// TIA Portal V17 export
// export: Created 2023-02-14T02:49:25.7164251Z, ExportSetting WithDefaults, DisplayName Totally Integrated Automation Portal, DisplayVersion V17, DisplayName TIA Portal Openness, DisplayVersion V17, DisplayName TIA Portal Teamcenter Gateway, DisplayVersion V17, DisplayName TIA Portal Version Control Interface, DisplayVersion V17, DisplayName SINAMICS Startdrive Advanced, DisplayVersion V17, DisplayName SINAMICS Startdrive G130, G150, S120, S150, SINAMICS MV, S210, DisplayVersion V17, DisplayName SINAMICS Startdrive G110M, G120, G120C, G120D, G120P, G115D, DisplayVersion V17, DisplayName STEP 7 Professional, DisplayVersion V17, DisplayName STEP 7 Safety, DisplayVersion V17, DisplayName WinCC Professional, DisplayVersion V17
FUNCTION_BLOCK "IO_Valve_Blend21"   // FB25, LAD
{ S7_Optimized_Access := 'FALSE' }
VERSION : 0.1
// stored: AutoNumber true, IsIECCheckEnabled false, SetENOAutomatically false, UDAEnableTagReadback false
   VAR_INPUT
      "lock 1" : Bool;
      "lock 2" : Bool;
      "lock 3" : Bool;
      "lock 4" : Bool;
      init : Bool;
      reset : Bool;
      testing : Bool;
   END_VAR
   VAR
      "AV-21.01" : "Valve";
      "AV-21.02" : "Valve";
      "AV-21.03" : "Valve";
      "AV-21.04" : "Valve";
      "AV-21.05" : "Valve";
      "AV-21.06" : "Valve";
      "AV-21.07" : "Valve";
      "AV-21.08" : "Valve";
      "AV-21.09" : "Valve";
      "AV-21.10" : "Valve";
      "AV-21.11" : "Valve";
      "AV-21.21" : "Valve";
      "AV-21.22" : "Valve";
      "AV-21.23" : "Valve";
      "AV-21.24" : "Valve";
      "AV-21.25" : "Valve";
      "AV-21.26" : "Valve";
      "AV-21.27" : "Valve";
      "AV-21.28" : "Valve";
      "AV-21.29" : "Valve";
      "AV-21.30" : "Valve";
      "AV-21.31" : "Valve";
      "AV-21.32" : "Valve";
      "AV-21.33" : "Valve";
      "AV-21.34" : "Valve";
      "AV-21.35" : "Valve";
      "AV-21.41" : "Valve";
      "AV-21.42" : "Valve";
   END_VAR
BEGIN

REGION Network 1 (SCL): FB OPEN AND CLOSE VALVE T-21
   IF #testing THEN
       // Statement section IF
       #"AV-21.01".FB_OPEN := #"AV-21.01".QCMD_OP;
       #"AV-21.01".FB_CLOSE := NOT #"AV-21.01".QCMD_OP;
       #"AV-21.02".FB_OPEN := #"AV-21.02".QCMD_OP;
       #"AV-21.02".FB_CLOSE := NOT #"AV-21.02".QCMD_OP;
       #"AV-21.03".FB_OPEN := #"AV-21.03".QCMD_OP;
       #"AV-21.03".FB_CLOSE := NOT #"AV-21.03".QCMD_OP;
       #"AV-21.04".FB_OPEN := #"AV-21.04".QCMD_OP;
       #"AV-21.04".FB_CLOSE := NOT #"AV-21.04".QCMD_OP;
       #"AV-21.05".FB_OPEN := #"AV-21.05".QCMD_OP;
       #"AV-21.05".FB_CLOSE := NOT #"AV-21.05".QCMD_OP;
       #"AV-21.06".FB_OPEN := #"AV-21.06".QCMD_OP;
       #"AV-21.06".FB_CLOSE := NOT #"AV-21.06".QCMD_OP;
       #"AV-21.07".FB_OPEN := #"AV-21.07".QCMD_OP;
       #"AV-21.07".FB_CLOSE := NOT #"AV-21.07".QCMD_OP;
       #"AV-21.08".FB_OPEN := #"AV-21.08".QCMD_OP;
       #"AV-21.08".FB_CLOSE := NOT #"AV-21.08".QCMD_OP;
       #"AV-21.09".FB_OPEN := #"AV-21.09".QCMD_OP;
       #"AV-21.09".FB_CLOSE := NOT #"AV-21.09".QCMD_OP;
       #"AV-21.10".FB_OPEN := #"AV-21.10".QCMD_OP;
       #"AV-21.10".FB_CLOSE := NOT #"AV-21.10".QCMD_OP;
       #"AV-21.11".FB_OPEN := #"AV-21.11".QCMD_OP;
       #"AV-21.11".FB_CLOSE := NOT #"AV-21.11".QCMD_OP;
       #"AV-21.21".FB_OPEN := #"AV-21.21".QCMD_OP;
       #"AV-21.21".FB_CLOSE := NOT #"AV-21.21".QCMD_OP;
       #"AV-21.22".FB_OPEN := #"AV-21.22".QCMD_OP;
       #"AV-21.22".FB_CLOSE := NOT #"AV-21.22".QCMD_OP;
       #"AV-21.23".FB_OPEN := #"AV-21.23".QCMD_OP;
       #"AV-21.23".FB_CLOSE := NOT #"AV-21.23".QCMD_OP;
       #"AV-21.24".FB_OPEN := #"AV-21.24".QCMD_OP;
       #"AV-21.24".FB_CLOSE := NOT #"AV-21.24".QCMD_OP;
       #"AV-21.25".FB_OPEN := #"AV-21.25".QCMD_OP;
       #"AV-21.25".FB_CLOSE := NOT #"AV-21.25".QCMD_OP;
       #"AV-21.26".FB_OPEN := #"AV-21.26".QCMD_OP;
       #"AV-21.26".FB_CLOSE := NOT #"AV-21.26".QCMD_OP;
       #"AV-21.27".FB_OPEN := #"AV-21.27".QCMD_OP;
       #"AV-21.27".FB_CLOSE := NOT #"AV-21.27".QCMD_OP;
       #"AV-21.28".FB_OPEN := #"AV-21.28".QCMD_OP;
       #"AV-21.28".FB_CLOSE := NOT #"AV-21.28".QCMD_OP;
       #"AV-21.29".FB_OPEN := #"AV-21.29".QCMD_OP;
       #"AV-21.29".FB_CLOSE := NOT #"AV-21.29".QCMD_OP;
       #"AV-21.30".FB_OPEN := #"AV-21.30".QCMD_OP;
       #"AV-21.30".FB_CLOSE := NOT #"AV-21.30".QCMD_OP;
       #"AV-21.31".FB_OPEN := #"AV-21.31".QCMD_OP;
       #"AV-21.31".FB_CLOSE := NOT #"AV-21.31".QCMD_OP;
       #"AV-21.32".FB_OPEN := #"AV-21.32".QCMD_OP;
       #"AV-21.32".FB_CLOSE := NOT #"AV-21.32".QCMD_OP;
       #"AV-21.33".FB_OPEN := #"AV-21.33".QCMD_OP;
       #"AV-21.33".FB_CLOSE := NOT #"AV-21.33".QCMD_OP;
       #"AV-21.34".FB_OPEN := #"AV-21.34".QCMD_OP;
       #"AV-21.34".FB_CLOSE := NOT #"AV-21.34".QCMD_OP;
       #"AV-21.35".FB_OPEN := #"AV-21.35".QCMD_OP;
       #"AV-21.35".FB_CLOSE := NOT #"AV-21.35".QCMD_OP;
       #"AV-21.41".FB_OPEN := #"AV-21.41".QCMD_OP;
       #"AV-21.41".FB_CLOSE := NOT #"AV-21.41".QCMD_OP;
       #"AV-21.42".FB_OPEN := #"AV-21.42".QCMD_OP;
       #"AV-21.42".FB_CLOSE := NOT #"AV-21.42".QCMD_OP;
   ELSE
       // Statement section ELSE
       #"AV-21.01".FB_OPEN := #"AV-21.01".QCMD_OP;
       #"AV-21.01".FB_CLOSE := NOT #"AV-21.01".QCMD_OP;
       #"AV-21.02".FB_OPEN := NOT "ZSC-21.02";
       #"AV-21.02".FB_CLOSE := "ZSC-21.02";
       #"AV-21.03".FB_OPEN := NOT "ZSC-21.03";
       #"AV-21.03".FB_CLOSE := "ZSC-21.03";
       #"AV-21.04".FB_OPEN := #"AV-21.04".QCMD_OP;
       #"AV-21.04".FB_CLOSE := NOT #"AV-21.04".QCMD_OP;
       #"AV-21.05".FB_OPEN := NOT "ZSC-21.05";
       #"AV-21.05".FB_CLOSE := "ZSC-21.05";
       #"AV-21.06".FB_OPEN := NOT "ZSC-21.06";
       #"AV-21.06".FB_CLOSE := "ZSC-21.06";
       #"AV-21.07".FB_OPEN := #"AV-21.07".QCMD_OP;
       #"AV-21.07".FB_CLOSE := NOT #"AV-21.07".QCMD_OP;
       #"AV-21.08".FB_OPEN := NOT "ZSC-21.08";
       #"AV-21.08".FB_CLOSE := "ZSC-21.08";
       #"AV-21.09".FB_OPEN := NOT "ZSC-21.09";
       #"AV-21.09".FB_CLOSE := "ZSC-21.09";
       #"AV-21.10".FB_OPEN := #"AV-21.10".QCMD_OP;
       #"AV-21.10".FB_CLOSE := NOT #"AV-21.10".QCMD_OP;
       #"AV-21.11".FB_OPEN := NOT "ZSC-21.11";
       #"AV-21.11".FB_CLOSE := "ZSC-21.11";
       #"AV-21.21".FB_OPEN := NOT "ZSC-21.21";
       #"AV-21.21".FB_CLOSE := "ZSC-21.21";
       #"AV-21.22".FB_OPEN := #"AV-21.22".QCMD_OP;
       #"AV-21.22".FB_CLOSE := NOT #"AV-21.22".QCMD_OP;
       #"AV-21.23".FB_OPEN := NOT "ZSC-21.23";
       #"AV-21.23".FB_CLOSE := "ZSC-21.23";
       #"AV-21.24".FB_OPEN := NOT "ZSC-21.24";
       #"AV-21.24".FB_CLOSE := "ZSC-21.24";
       #"AV-21.25".FB_OPEN := NOT "ZSC-21.25";
       #"AV-21.25".FB_CLOSE := "ZSC-21.25";
       #"AV-21.26".FB_OPEN := #"AV-21.26".QCMD_OP;
       #"AV-21.26".FB_CLOSE := NOT #"AV-21.26".QCMD_OP;
       #"AV-21.27".FB_OPEN := NOT "ZSC-21.27";
       #"AV-21.27".FB_CLOSE := "ZSC-21.27";
       #"AV-21.28".FB_OPEN := NOT "ZSC-21.28";
       #"AV-21.28".FB_CLOSE := "ZSC-21.28";
       #"AV-21.29".FB_OPEN := #"AV-21.29".QCMD_OP;
       #"AV-21.29".FB_CLOSE := NOT #"AV-21.29".QCMD_OP;
       #"AV-21.30".FB_OPEN := #"AV-21.30".QCMD_OP;
       #"AV-21.30".FB_CLOSE := NOT #"AV-21.30".QCMD_OP;
       #"AV-21.31".FB_OPEN := NOT "ZSC-21.31";
       #"AV-21.31".FB_CLOSE := "ZSC-21.31";
       #"AV-21.32".FB_OPEN := NOT "ZSC-21.32";
       #"AV-21.32".FB_CLOSE := "ZSC-21.32";
       #"AV-21.33".FB_OPEN := NOT "ZSC-21.33";
       #"AV-21.33".FB_CLOSE := "ZSC-21.33";
       #"AV-21.34".FB_OPEN := NOT "ZSC-21.34";
       #"AV-21.34".FB_CLOSE := "ZSC-21.34";
       #"AV-21.35".FB_OPEN := NOT "ZSC-21.35";
       #"AV-21.35".FB_CLOSE := "ZSC-21.35";
       #"AV-21.41".FB_OPEN := #"AV-21.41".QCMD_OP;
       #"AV-21.41".FB_CLOSE := NOT #"AV-21.41".QCMD_OP;
       #"AV-21.42".FB_OPEN := #"AV-21.42".QCMD_OP;
       #"AV-21.42".FB_CLOSE := NOT #"AV-21.42".QCMD_OP;
   END_IF;
END_REGION

NETWORK
TITLE = FB MONITORING TIME VALVE T-21
// FB OPEN TIME
      L     T#20s;
      T     #"AV-21.01".MON_T;
      T     #"AV-21.02".MON_T;
      T     #"AV-21.03".MON_T;
      T     #"AV-21.04".MON_T;
      T     #"AV-21.05".MON_T;
      T     #"AV-21.06".MON_T;
      T     #"AV-21.07".MON_T;
      T     #"AV-21.08".MON_T;
      T     #"AV-21.09".MON_T;
      T     #"AV-21.10".MON_T;
      T     #"AV-21.11".MON_T;
      T     #"AV-21.21".MON_T;
      T     #"AV-21.22".MON_T;
      T     #"AV-21.23".MON_T;
      T     #"AV-21.24".MON_T;
      T     #"AV-21.25".MON_T;
      T     #"AV-21.26".MON_T;
      T     #"AV-21.27".MON_T;
      T     #"AV-21.28".MON_T;
      T     #"AV-21.29".MON_T;
      T     #"AV-21.30".MON_T;
      T     #"AV-21.31".MON_T;
      T     #"AV-21.32".MON_T;
      T     #"AV-21.33".MON_T;
      T     #"AV-21.34".MON_T;
      T     #"AV-21.35".MON_T;
      T     #"AV-21.41".MON_T;
      T     #"AV-21.42".MON_T;

// FB CLOSE TIME
      L     T#20s;
      T     #"AV-21.01".MON_T_CLOSE;
      T     #"AV-21.02".MON_T_CLOSE;
      T     #"AV-21.03".MON_T_CLOSE;
      T     #"AV-21.04".MON_T_CLOSE;
      T     #"AV-21.05".MON_T_CLOSE;
      T     #"AV-21.06".MON_T_CLOSE;
      T     #"AV-21.07".MON_T_CLOSE;
      T     #"AV-21.08".MON_T_CLOSE;
      T     #"AV-21.09".MON_T_CLOSE;
      T     #"AV-21.10".MON_T_CLOSE;
      T     #"AV-21.11".MON_T_CLOSE;
      T     #"AV-21.21".MON_T_CLOSE;
      T     #"AV-21.22".MON_T_CLOSE;
      T     #"AV-21.23".MON_T_CLOSE;
      T     #"AV-21.24".MON_T_CLOSE;
      T     #"AV-21.25".MON_T_CLOSE;
      T     #"AV-21.26".MON_T_CLOSE;
      T     #"AV-21.27".MON_T_CLOSE;
      T     #"AV-21.28".MON_T_CLOSE;
      T     #"AV-21.29".MON_T_CLOSE;
      T     #"AV-21.30".MON_T_CLOSE;
      T     #"AV-21.31".MON_T_CLOSE;
      T     #"AV-21.32".MON_T_CLOSE;
      T     #"AV-21.33".MON_T_CLOSE;
      T     #"AV-21.34".MON_T_CLOSE;
      T     #"AV-21.35".MON_T_CLOSE;
      T     #"AV-21.41".MON_T_CLOSE;
      T     #"AV-21.42".MON_T_CLOSE;


REGION Network 3: AV-21.01
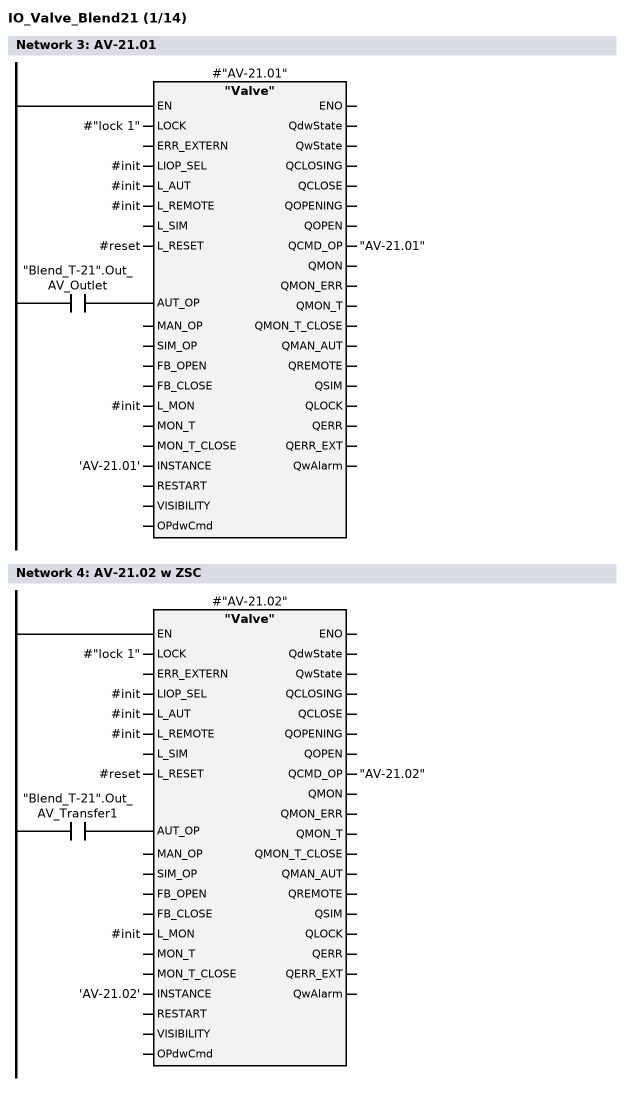
   RUNG wire#powerrail
      #"AV-21.01"(AUT_OP := wire#w1, LOCK := #"lock 1", ERR_EXTERN :=, LIOP_SEL := #init, L_AUT := #init, L_REMOTE := #init, L_SIM :=, L_RESET := #reset, MAN_OP :=, SIM_OP :=, FB_OPEN :=, FB_CLOSE :=, L_MON := #init, MON_T :=, MON_T_CLOSE :=, INSTANCE := 'AV-21.01', RESTART :=, VISIBILITY :=, OPdwCmd :=, QdwState =>, QwState =>, QCLOSING =>, QCLOSE =>, QOPENING =>, QOPEN =>, QCMD_OP => "AV-21.01", QMON =>, QMON_ERR =>, QMON_T =>, QMON_T_CLOSE =>, QMAN_AUT =>, QREMOTE =>, QSIM =>, QLOCK =>, QERR =>, QERR_EXT =>, QwAlarm =>)
   END_RUNG
   RUNG wire#powerrail
      Contact( "Blend_T-21".Out_AV_Outlet )
   END_RUNG wire#w1
   // the same network as SCL:
   #"AV-21.01"(LOCK := #"lock 1",   // "Valve"
               LIOP_SEL := #init,
               L_AUT := #init,
               L_REMOTE := #init,
               L_RESET := #reset,
               AUT_OP := "Blend_T-21".Out_AV_Outlet,
               L_MON := #init,
               INSTANCE := 'AV-21.01',
               QCMD_OP => "AV-21.01");
END_REGION

REGION Network 4: AV-21.02 w ZSC
   RUNG wire#powerrail
      #"AV-21.02"(AUT_OP := wire#w1, LOCK := #"lock 1", ERR_EXTERN :=, LIOP_SEL := #init, L_AUT := #init, L_REMOTE := #init, L_SIM :=, L_RESET := #reset, MAN_OP :=, SIM_OP :=, FB_OPEN :=, FB_CLOSE :=, L_MON := #init, MON_T :=, MON_T_CLOSE :=, INSTANCE := 'AV-21.02', RESTART :=, VISIBILITY :=, OPdwCmd :=, QdwState =>, QwState =>, QCLOSING =>, QCLOSE =>, QOPENING =>, QOPEN =>, QCMD_OP => "AV-21.02", QMON =>, QMON_ERR =>, QMON_T =>, QMON_T_CLOSE =>, QMAN_AUT =>, QREMOTE =>, QSIM =>, QLOCK =>, QERR =>, QERR_EXT =>, QwAlarm =>)
   END_RUNG
   RUNG wire#powerrail
      Contact( "Blend_T-21".Out_AV_Transfer1 )
   END_RUNG wire#w1
   // the same network as SCL:
   #"AV-21.02"(LOCK := #"lock 1",   // "Valve"
               LIOP_SEL := #init,
               L_AUT := #init,
               L_REMOTE := #init,
               L_RESET := #reset,
               AUT_OP := "Blend_T-21".Out_AV_Transfer1,
               L_MON := #init,
               INSTANCE := 'AV-21.02',
               QCMD_OP => "AV-21.02");
END_REGION

REGION Network 5: AV-21.03 w ZSC
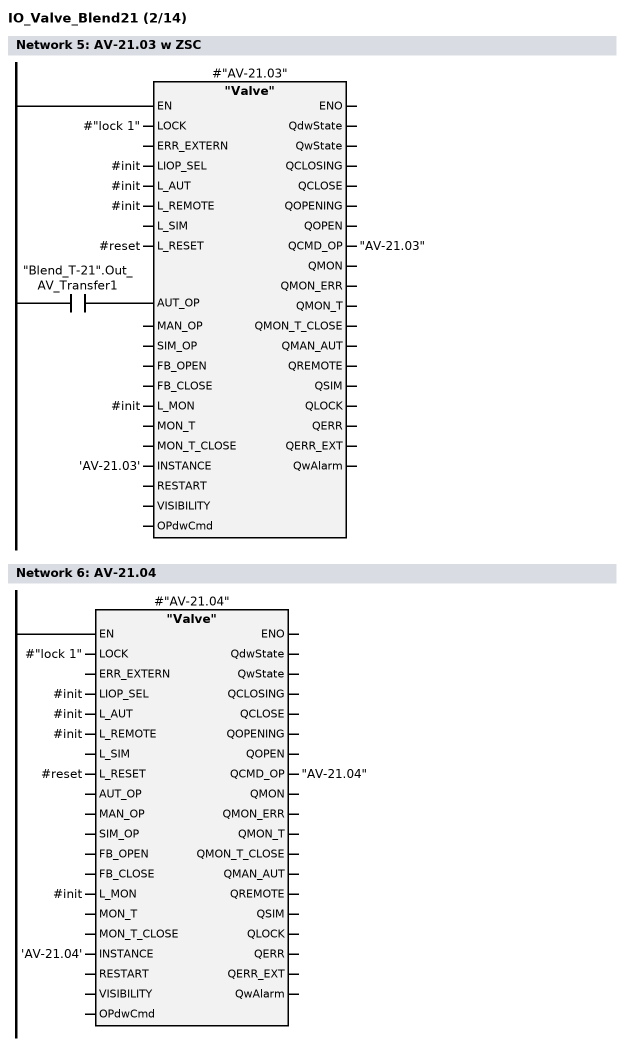
   RUNG wire#powerrail
      #"AV-21.03"(AUT_OP := wire#w1, LOCK := #"lock 1", ERR_EXTERN :=, LIOP_SEL := #init, L_AUT := #init, L_REMOTE := #init, L_SIM :=, L_RESET := #reset, MAN_OP :=, SIM_OP :=, FB_OPEN :=, FB_CLOSE :=, L_MON := #init, MON_T :=, MON_T_CLOSE :=, INSTANCE := 'AV-21.03', RESTART :=, VISIBILITY :=, OPdwCmd :=, QdwState =>, QwState =>, QCLOSING =>, QCLOSE =>, QOPENING =>, QOPEN =>, QCMD_OP => "AV-21.03", QMON =>, QMON_ERR =>, QMON_T =>, QMON_T_CLOSE =>, QMAN_AUT =>, QREMOTE =>, QSIM =>, QLOCK =>, QERR =>, QERR_EXT =>, QwAlarm =>)
   END_RUNG
   RUNG wire#powerrail
      Contact( "Blend_T-21".Out_AV_Transfer1 )
   END_RUNG wire#w1
   // the same network as SCL:
   #"AV-21.03"(LOCK := #"lock 1",   // "Valve"
               LIOP_SEL := #init,
               L_AUT := #init,
               L_REMOTE := #init,
               L_RESET := #reset,
               AUT_OP := "Blend_T-21".Out_AV_Transfer1,
               L_MON := #init,
               INSTANCE := 'AV-21.03',
               QCMD_OP => "AV-21.03");
END_REGION

REGION Network 6: AV-21.04
   RUNG wire#powerrail
      #"AV-21.04"(LOCK := #"lock 1", ERR_EXTERN :=, LIOP_SEL := #init, L_AUT := #init, L_REMOTE := #init, L_SIM :=, L_RESET := #reset, AUT_OP :=, MAN_OP :=, SIM_OP :=, FB_OPEN :=, FB_CLOSE :=, L_MON := #init, MON_T :=, MON_T_CLOSE :=, INSTANCE := 'AV-21.04', RESTART :=, VISIBILITY :=, OPdwCmd :=, QdwState =>, QwState =>, QCLOSING =>, QCLOSE =>, QOPENING =>, QOPEN =>, QCMD_OP => "AV-21.04", QMON =>, QMON_ERR =>, QMON_T =>, QMON_T_CLOSE =>, QMAN_AUT =>, QREMOTE =>, QSIM =>, QLOCK =>, QERR =>, QERR_EXT =>, QwAlarm =>)
   END_RUNG
   // the same network as SCL:
   #"AV-21.04"(LOCK := #"lock 1",   // "Valve"
               LIOP_SEL := #init,
               L_AUT := #init,
               L_REMOTE := #init,
               L_RESET := #reset,
               L_MON := #init,
               INSTANCE := 'AV-21.04',
               QCMD_OP => "AV-21.04");
END_REGION

REGION Network 7: AV-21.05 w ZSC
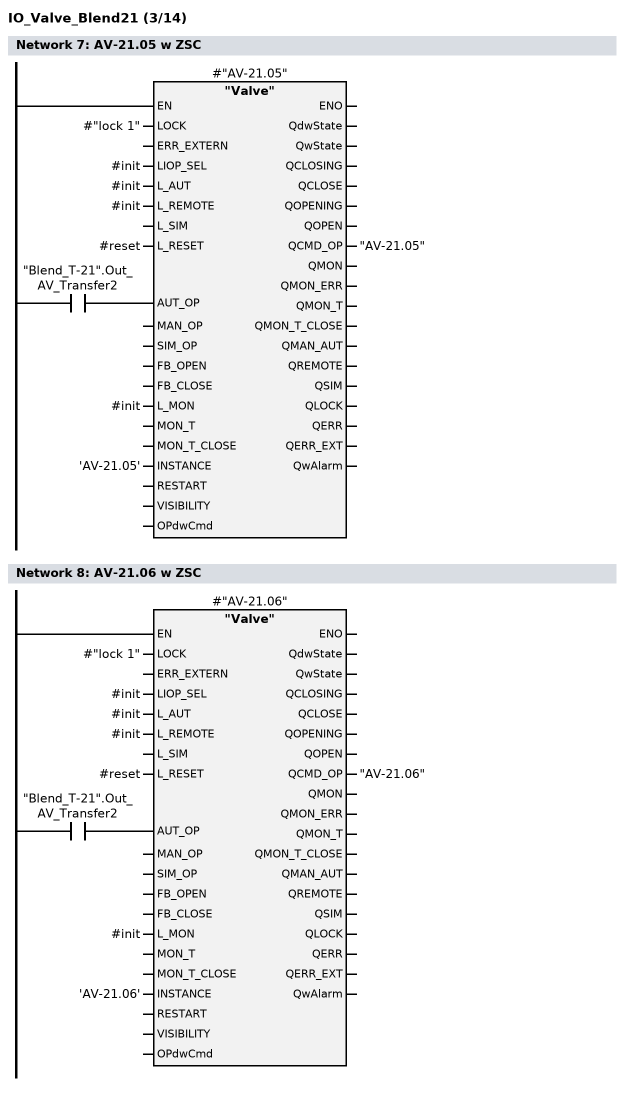
   RUNG wire#powerrail
      #"AV-21.05"(AUT_OP := wire#w1, LOCK := #"lock 1", ERR_EXTERN :=, LIOP_SEL := #init, L_AUT := #init, L_REMOTE := #init, L_SIM :=, L_RESET := #reset, MAN_OP :=, SIM_OP :=, FB_OPEN :=, FB_CLOSE :=, L_MON := #init, MON_T :=, MON_T_CLOSE :=, INSTANCE := 'AV-21.05', RESTART :=, VISIBILITY :=, OPdwCmd :=, QdwState =>, QwState =>, QCLOSING =>, QCLOSE =>, QOPENING =>, QOPEN =>, QCMD_OP => "AV-21.05", QMON =>, QMON_ERR =>, QMON_T =>, QMON_T_CLOSE =>, QMAN_AUT =>, QREMOTE =>, QSIM =>, QLOCK =>, QERR =>, QERR_EXT =>, QwAlarm =>)
   END_RUNG
   RUNG wire#powerrail
      Contact( "Blend_T-21".Out_AV_Transfer2 )
   END_RUNG wire#w1
   // the same network as SCL:
   #"AV-21.05"(LOCK := #"lock 1",   // "Valve"
               LIOP_SEL := #init,
               L_AUT := #init,
               L_REMOTE := #init,
               L_RESET := #reset,
               AUT_OP := "Blend_T-21".Out_AV_Transfer2,
               L_MON := #init,
               INSTANCE := 'AV-21.05',
               QCMD_OP => "AV-21.05");
END_REGION

REGION Network 8: AV-21.06 w ZSC
   RUNG wire#powerrail
      #"AV-21.06"(AUT_OP := wire#w1, LOCK := #"lock 1", ERR_EXTERN :=, LIOP_SEL := #init, L_AUT := #init, L_REMOTE := #init, L_SIM :=, L_RESET := #reset, MAN_OP :=, SIM_OP :=, FB_OPEN :=, FB_CLOSE :=, L_MON := #init, MON_T :=, MON_T_CLOSE :=, INSTANCE := 'AV-21.06', RESTART :=, VISIBILITY :=, OPdwCmd :=, QdwState =>, QwState =>, QCLOSING =>, QCLOSE =>, QOPENING =>, QOPEN =>, QCMD_OP => "AV-21.06", QMON =>, QMON_ERR =>, QMON_T =>, QMON_T_CLOSE =>, QMAN_AUT =>, QREMOTE =>, QSIM =>, QLOCK =>, QERR =>, QERR_EXT =>, QwAlarm =>)
   END_RUNG
   RUNG wire#powerrail
      Contact( "Blend_T-21".Out_AV_Transfer2 )
   END_RUNG wire#w1
   // the same network as SCL:
   #"AV-21.06"(LOCK := #"lock 1",   // "Valve"
               LIOP_SEL := #init,
               L_AUT := #init,
               L_REMOTE := #init,
               L_RESET := #reset,
               AUT_OP := "Blend_T-21".Out_AV_Transfer2,
               L_MON := #init,
               INSTANCE := 'AV-21.06',
               QCMD_OP => "AV-21.06");
END_REGION

REGION Network 9: AV-21.07
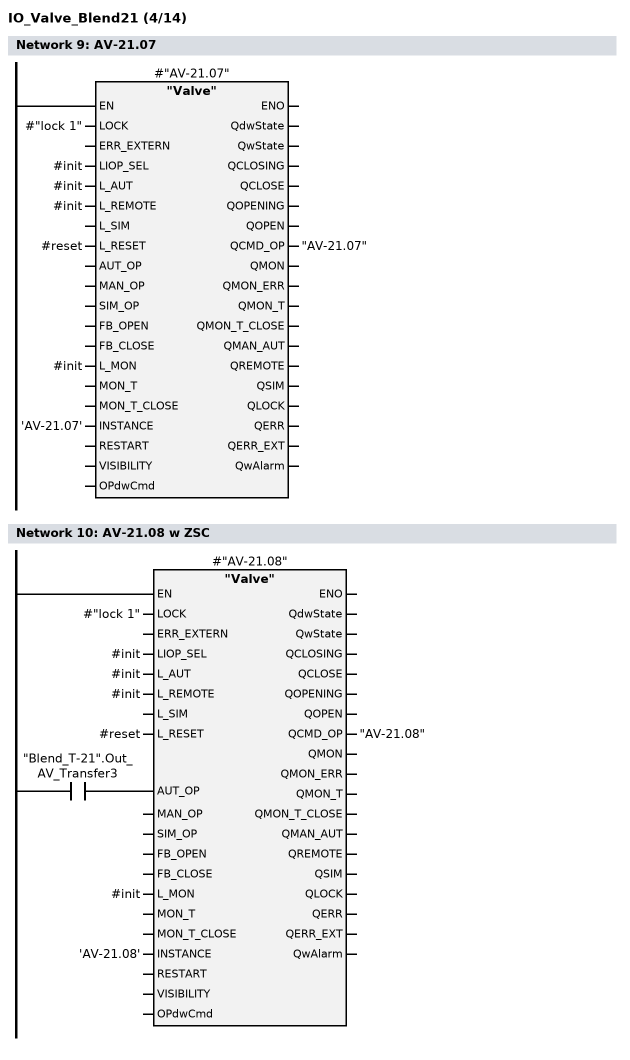
   RUNG wire#powerrail
      #"AV-21.07"(LOCK := #"lock 1", ERR_EXTERN :=, LIOP_SEL := #init, L_AUT := #init, L_REMOTE := #init, L_SIM :=, L_RESET := #reset, AUT_OP :=, MAN_OP :=, SIM_OP :=, FB_OPEN :=, FB_CLOSE :=, L_MON := #init, MON_T :=, MON_T_CLOSE :=, INSTANCE := 'AV-21.07', RESTART :=, VISIBILITY :=, OPdwCmd :=, QdwState =>, QwState =>, QCLOSING =>, QCLOSE =>, QOPENING =>, QOPEN =>, QCMD_OP => "AV-21.07", QMON =>, QMON_ERR =>, QMON_T =>, QMON_T_CLOSE =>, QMAN_AUT =>, QREMOTE =>, QSIM =>, QLOCK =>, QERR =>, QERR_EXT =>, QwAlarm =>)
   END_RUNG
   // the same network as SCL:
   #"AV-21.07"(LOCK := #"lock 1",   // "Valve"
               LIOP_SEL := #init,
               L_AUT := #init,
               L_REMOTE := #init,
               L_RESET := #reset,
               L_MON := #init,
               INSTANCE := 'AV-21.07',
               QCMD_OP => "AV-21.07");
END_REGION

REGION Network 10: AV-21.08 w ZSC
   RUNG wire#powerrail
      #"AV-21.08"(AUT_OP := wire#w1, LOCK := #"lock 1", ERR_EXTERN :=, LIOP_SEL := #init, L_AUT := #init, L_REMOTE := #init, L_SIM :=, L_RESET := #reset, MAN_OP :=, SIM_OP :=, FB_OPEN :=, FB_CLOSE :=, L_MON := #init, MON_T :=, MON_T_CLOSE :=, INSTANCE := 'AV-21.08', RESTART :=, VISIBILITY :=, OPdwCmd :=, QdwState =>, QwState =>, QCLOSING =>, QCLOSE =>, QOPENING =>, QOPEN =>, QCMD_OP => "AV-21.08", QMON =>, QMON_ERR =>, QMON_T =>, QMON_T_CLOSE =>, QMAN_AUT =>, QREMOTE =>, QSIM =>, QLOCK =>, QERR =>, QERR_EXT =>, QwAlarm =>)
   END_RUNG
   RUNG wire#powerrail
      Contact( "Blend_T-21".Out_AV_Transfer3 )
   END_RUNG wire#w1
   // the same network as SCL:
   #"AV-21.08"(LOCK := #"lock 1",   // "Valve"
               LIOP_SEL := #init,
               L_AUT := #init,
               L_REMOTE := #init,
               L_RESET := #reset,
               AUT_OP := "Blend_T-21".Out_AV_Transfer3,
               L_MON := #init,
               INSTANCE := 'AV-21.08',
               QCMD_OP => "AV-21.08");
END_REGION

REGION Network 11: AV-21.09 w ZSC
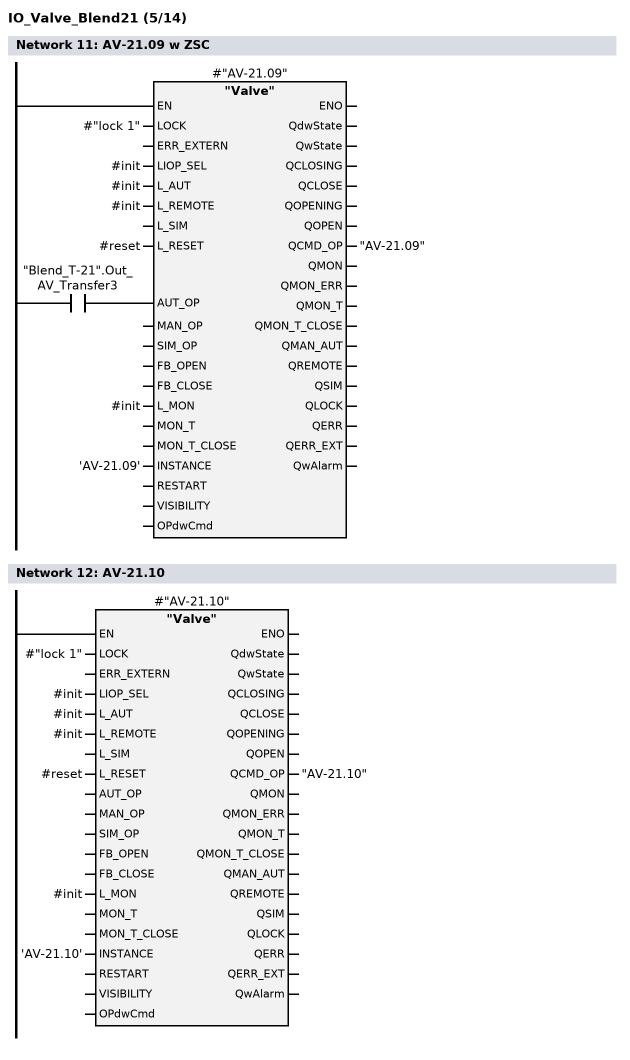
   RUNG wire#powerrail
      #"AV-21.09"(AUT_OP := wire#w1, LOCK := #"lock 1", ERR_EXTERN :=, LIOP_SEL := #init, L_AUT := #init, L_REMOTE := #init, L_SIM :=, L_RESET := #reset, MAN_OP :=, SIM_OP :=, FB_OPEN :=, FB_CLOSE :=, L_MON := #init, MON_T :=, MON_T_CLOSE :=, INSTANCE := 'AV-21.09', RESTART :=, VISIBILITY :=, OPdwCmd :=, QdwState =>, QwState =>, QCLOSING =>, QCLOSE =>, QOPENING =>, QOPEN =>, QCMD_OP => "AV-21.09", QMON =>, QMON_ERR =>, QMON_T =>, QMON_T_CLOSE =>, QMAN_AUT =>, QREMOTE =>, QSIM =>, QLOCK =>, QERR =>, QERR_EXT =>, QwAlarm =>)
   END_RUNG
   RUNG wire#powerrail
      Contact( "Blend_T-21".Out_AV_Transfer3 )
   END_RUNG wire#w1
   // the same network as SCL:
   #"AV-21.09"(LOCK := #"lock 1",   // "Valve"
               LIOP_SEL := #init,
               L_AUT := #init,
               L_REMOTE := #init,
               L_RESET := #reset,
               AUT_OP := "Blend_T-21".Out_AV_Transfer3,
               L_MON := #init,
               INSTANCE := 'AV-21.09',
               QCMD_OP => "AV-21.09");
END_REGION

REGION Network 12: AV-21.10
   RUNG wire#powerrail
      #"AV-21.10"(LOCK := #"lock 1", ERR_EXTERN :=, LIOP_SEL := #init, L_AUT := #init, L_REMOTE := #init, L_SIM :=, L_RESET := #reset, AUT_OP :=, MAN_OP :=, SIM_OP :=, FB_OPEN :=, FB_CLOSE :=, L_MON := #init, MON_T :=, MON_T_CLOSE :=, INSTANCE := 'AV-21.10', RESTART :=, VISIBILITY :=, OPdwCmd :=, QdwState =>, QwState =>, QCLOSING =>, QCLOSE =>, QOPENING =>, QOPEN =>, QCMD_OP => "AV-21.10", QMON =>, QMON_ERR =>, QMON_T =>, QMON_T_CLOSE =>, QMAN_AUT =>, QREMOTE =>, QSIM =>, QLOCK =>, QERR =>, QERR_EXT =>, QwAlarm =>)
   END_RUNG
   // the same network as SCL:
   #"AV-21.10"(LOCK := #"lock 1",   // "Valve"
               LIOP_SEL := #init,
               L_AUT := #init,
               L_REMOTE := #init,
               L_RESET := #reset,
               L_MON := #init,
               INSTANCE := 'AV-21.10',
               QCMD_OP => "AV-21.10");
END_REGION

REGION Network 13: AV-21.11 w ZSC
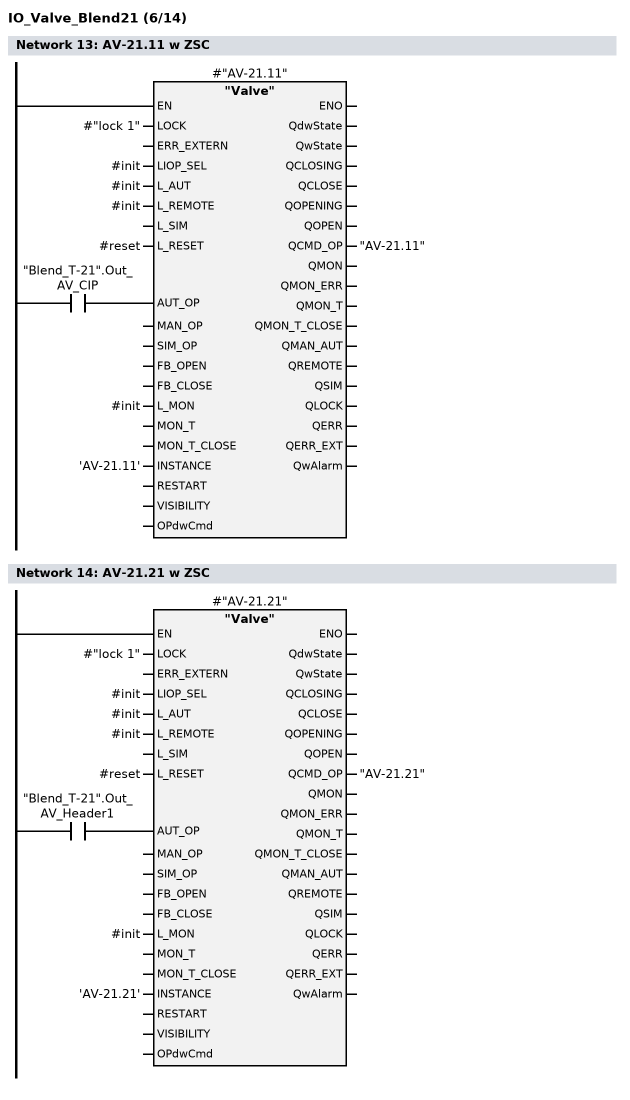
   RUNG wire#powerrail
      #"AV-21.11"(AUT_OP := wire#w1, LOCK := #"lock 1", ERR_EXTERN :=, LIOP_SEL := #init, L_AUT := #init, L_REMOTE := #init, L_SIM :=, L_RESET := #reset, MAN_OP :=, SIM_OP :=, FB_OPEN :=, FB_CLOSE :=, L_MON := #init, MON_T :=, MON_T_CLOSE :=, INSTANCE := 'AV-21.11', RESTART :=, VISIBILITY :=, OPdwCmd :=, QdwState =>, QwState =>, QCLOSING =>, QCLOSE =>, QOPENING =>, QOPEN =>, QCMD_OP => "AV-21.11", QMON =>, QMON_ERR =>, QMON_T =>, QMON_T_CLOSE =>, QMAN_AUT =>, QREMOTE =>, QSIM =>, QLOCK =>, QERR =>, QERR_EXT =>, QwAlarm =>)
   END_RUNG
   RUNG wire#powerrail
      Contact( "Blend_T-21".Out_AV_CIP )
   END_RUNG wire#w1
   // the same network as SCL:
   #"AV-21.11"(LOCK := #"lock 1",   // "Valve"
               LIOP_SEL := #init,
               L_AUT := #init,
               L_REMOTE := #init,
               L_RESET := #reset,
               AUT_OP := "Blend_T-21".Out_AV_CIP,
               L_MON := #init,
               INSTANCE := 'AV-21.11',
               QCMD_OP => "AV-21.11");
END_REGION

REGION Network 14: AV-21.21 w ZSC
   RUNG wire#powerrail
      #"AV-21.21"(AUT_OP := wire#w1, LOCK := #"lock 1", ERR_EXTERN :=, LIOP_SEL := #init, L_AUT := #init, L_REMOTE := #init, L_SIM :=, L_RESET := #reset, MAN_OP :=, SIM_OP :=, FB_OPEN :=, FB_CLOSE :=, L_MON := #init, MON_T :=, MON_T_CLOSE :=, INSTANCE := 'AV-21.21', RESTART :=, VISIBILITY :=, OPdwCmd :=, QdwState =>, QwState =>, QCLOSING =>, QCLOSE =>, QOPENING =>, QOPEN =>, QCMD_OP => "AV-21.21", QMON =>, QMON_ERR =>, QMON_T =>, QMON_T_CLOSE =>, QMAN_AUT =>, QREMOTE =>, QSIM =>, QLOCK =>, QERR =>, QERR_EXT =>, QwAlarm =>)
   END_RUNG
   RUNG wire#powerrail
      Contact( "Blend_T-21".Out_AV_Header1 )
   END_RUNG wire#w1
   // the same network as SCL:
   #"AV-21.21"(LOCK := #"lock 1",   // "Valve"
               LIOP_SEL := #init,
               L_AUT := #init,
               L_REMOTE := #init,
               L_RESET := #reset,
               AUT_OP := "Blend_T-21".Out_AV_Header1,
               L_MON := #init,
               INSTANCE := 'AV-21.21',
               QCMD_OP => "AV-21.21");
END_REGION

REGION Network 15: AV-21.22
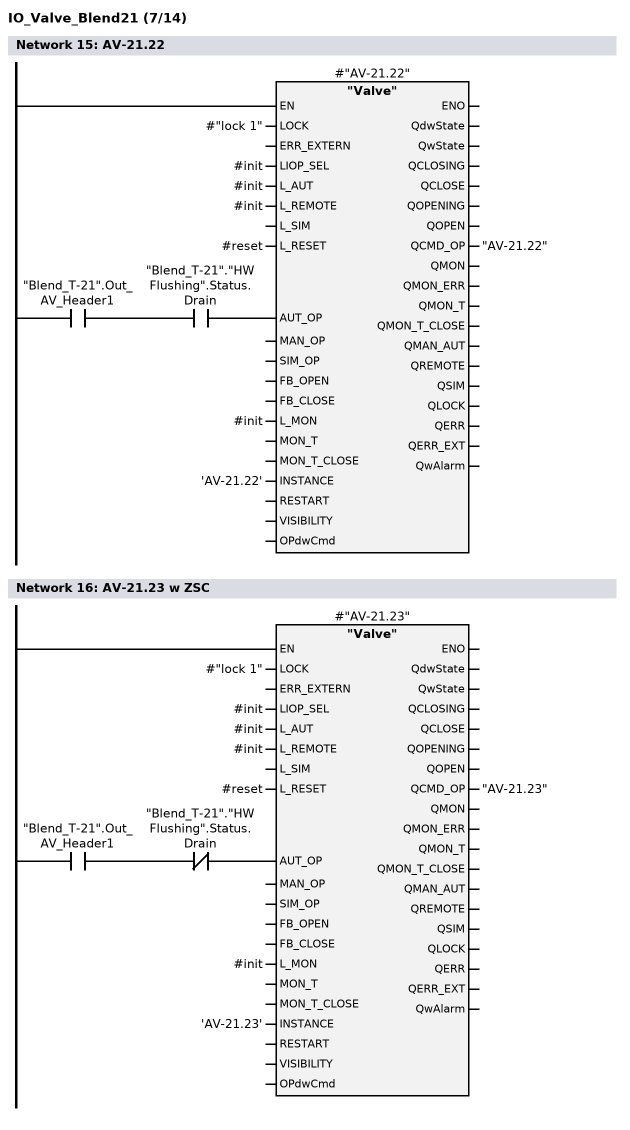
   RUNG wire#powerrail
      #"AV-21.22"(AUT_OP := wire#w1, LOCK := #"lock 1", ERR_EXTERN :=, LIOP_SEL := #init, L_AUT := #init, L_REMOTE := #init, L_SIM :=, L_RESET := #reset, MAN_OP :=, SIM_OP :=, FB_OPEN :=, FB_CLOSE :=, L_MON := #init, MON_T :=, MON_T_CLOSE :=, INSTANCE := 'AV-21.22', RESTART :=, VISIBILITY :=, OPdwCmd :=, QdwState =>, QwState =>, QCLOSING =>, QCLOSE =>, QOPENING =>, QOPEN =>, QCMD_OP => "AV-21.22", QMON =>, QMON_ERR =>, QMON_T =>, QMON_T_CLOSE =>, QMAN_AUT =>, QREMOTE =>, QSIM =>, QLOCK =>, QERR =>, QERR_EXT =>, QwAlarm =>)
   END_RUNG
   RUNG wire#powerrail
      Contact( "Blend_T-21".Out_AV_Header1 )
      Contact( "Blend_T-21"."HW Flushing".Status.Drain )
   END_RUNG wire#w1
   // the same network as SCL:
   #"AV-21.22"(LOCK := #"lock 1",   // "Valve"
               LIOP_SEL := #init,
               L_AUT := #init,
               L_REMOTE := #init,
               L_RESET := #reset,
               AUT_OP := "Blend_T-21".Out_AV_Header1 AND "Blend_T-21"."HW Flushing".Status.Drain,
               L_MON := #init,
               INSTANCE := 'AV-21.22',
               QCMD_OP => "AV-21.22");
END_REGION

REGION Network 16: AV-21.23 w ZSC
   RUNG wire#powerrail
      #"AV-21.23"(AUT_OP := wire#w1, LOCK := #"lock 1", ERR_EXTERN :=, LIOP_SEL := #init, L_AUT := #init, L_REMOTE := #init, L_SIM :=, L_RESET := #reset, MAN_OP :=, SIM_OP :=, FB_OPEN :=, FB_CLOSE :=, L_MON := #init, MON_T :=, MON_T_CLOSE :=, INSTANCE := 'AV-21.23', RESTART :=, VISIBILITY :=, OPdwCmd :=, QdwState =>, QwState =>, QCLOSING =>, QCLOSE =>, QOPENING =>, QOPEN =>, QCMD_OP => "AV-21.23", QMON =>, QMON_ERR =>, QMON_T =>, QMON_T_CLOSE =>, QMAN_AUT =>, QREMOTE =>, QSIM =>, QLOCK =>, QERR =>, QERR_EXT =>, QwAlarm =>)
   END_RUNG
   RUNG wire#powerrail
      Contact( "Blend_T-21".Out_AV_Header1 )
      I_Contact( "Blend_T-21"."HW Flushing".Status.Drain )
   END_RUNG wire#w1
   // the same network as SCL:
   #"AV-21.23"(LOCK := #"lock 1",   // "Valve"
               LIOP_SEL := #init,
               L_AUT := #init,
               L_REMOTE := #init,
               L_RESET := #reset,
               AUT_OP := "Blend_T-21".Out_AV_Header1 AND NOT "Blend_T-21"."HW Flushing".Status.Drain,
               L_MON := #init,
               INSTANCE := 'AV-21.23',
               QCMD_OP => "AV-21.23");
END_REGION

REGION Network 17: AV-21.24 w ZSC
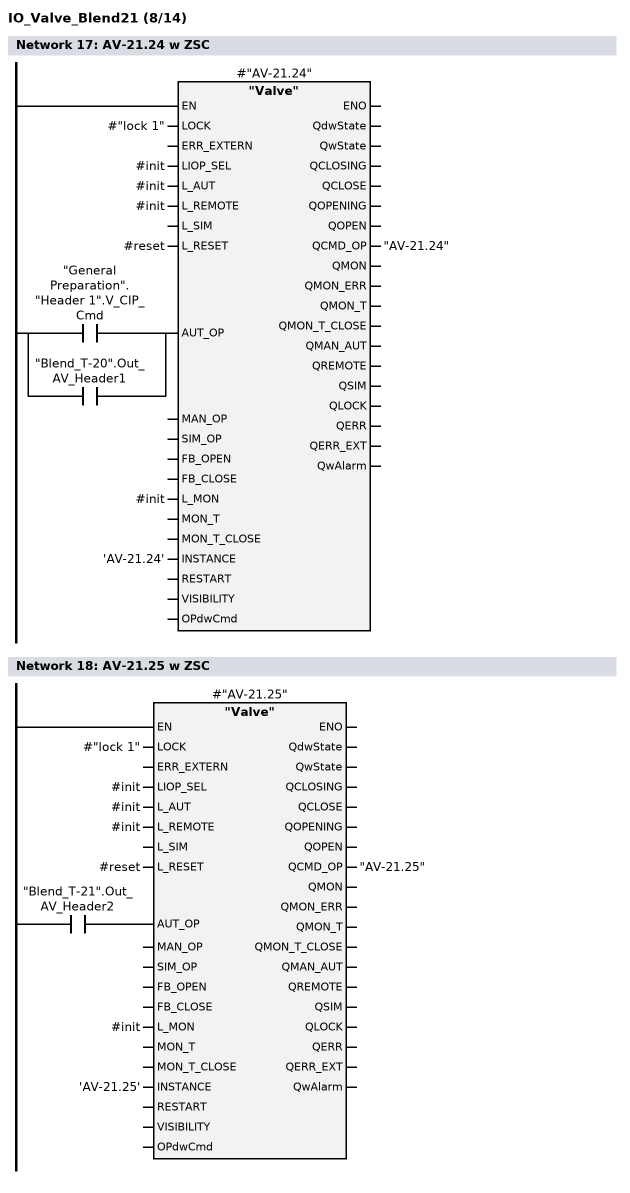
   RUNG wire#powerrail
      #"AV-21.24"(AUT_OP := wire#w1, LOCK := #"lock 1", ERR_EXTERN :=, LIOP_SEL := #init, L_AUT := #init, L_REMOTE := #init, L_SIM :=, L_RESET := #reset, MAN_OP :=, SIM_OP :=, FB_OPEN :=, FB_CLOSE :=, L_MON := #init, MON_T :=, MON_T_CLOSE :=, INSTANCE := 'AV-21.24', RESTART :=, VISIBILITY :=, OPdwCmd :=, QdwState =>, QwState =>, QCLOSING =>, QCLOSE =>, QOPENING =>, QOPEN =>, QCMD_OP => "AV-21.24", QMON =>, QMON_ERR =>, QMON_T =>, QMON_T_CLOSE =>, QMAN_AUT =>, QREMOTE =>, QSIM =>, QLOCK =>, QERR =>, QERR_EXT =>, QwAlarm =>)
   END_RUNG
   RUNG wire#powerrail
      Contact( "General Preparation"."Header 1".V_CIP_Cmd )
   END_RUNG wire#w1
   RUNG wire#powerrail
      Contact( "Blend_T-20".Out_AV_Header1 )
   END_RUNG wire#w1
   // the same network as SCL:
   #"AV-21.24"(LOCK := #"lock 1",   // "Valve"
               LIOP_SEL := #init,
               L_AUT := #init,
               L_REMOTE := #init,
               L_RESET := #reset,
               AUT_OP := "General Preparation"."Header 1".V_CIP_Cmd OR "Blend_T-20".Out_AV_Header1,
               L_MON := #init,
               INSTANCE := 'AV-21.24',
               QCMD_OP => "AV-21.24");
END_REGION

REGION Network 18: AV-21.25 w ZSC
   RUNG wire#powerrail
      #"AV-21.25"(AUT_OP := wire#w1, LOCK := #"lock 1", ERR_EXTERN :=, LIOP_SEL := #init, L_AUT := #init, L_REMOTE := #init, L_SIM :=, L_RESET := #reset, MAN_OP :=, SIM_OP :=, FB_OPEN :=, FB_CLOSE :=, L_MON := #init, MON_T :=, MON_T_CLOSE :=, INSTANCE := 'AV-21.25', RESTART :=, VISIBILITY :=, OPdwCmd :=, QdwState =>, QwState =>, QCLOSING =>, QCLOSE =>, QOPENING =>, QOPEN =>, QCMD_OP => "AV-21.25", QMON =>, QMON_ERR =>, QMON_T =>, QMON_T_CLOSE =>, QMAN_AUT =>, QREMOTE =>, QSIM =>, QLOCK =>, QERR =>, QERR_EXT =>, QwAlarm =>)
   END_RUNG
   RUNG wire#powerrail
      Contact( "Blend_T-21".Out_AV_Header2 )
   END_RUNG wire#w1
   // the same network as SCL:
   #"AV-21.25"(LOCK := #"lock 1",   // "Valve"
               LIOP_SEL := #init,
               L_AUT := #init,
               L_REMOTE := #init,
               L_RESET := #reset,
               AUT_OP := "Blend_T-21".Out_AV_Header2,
               L_MON := #init,
               INSTANCE := 'AV-21.25',
               QCMD_OP => "AV-21.25");
END_REGION

REGION Network 19: AV-21.26
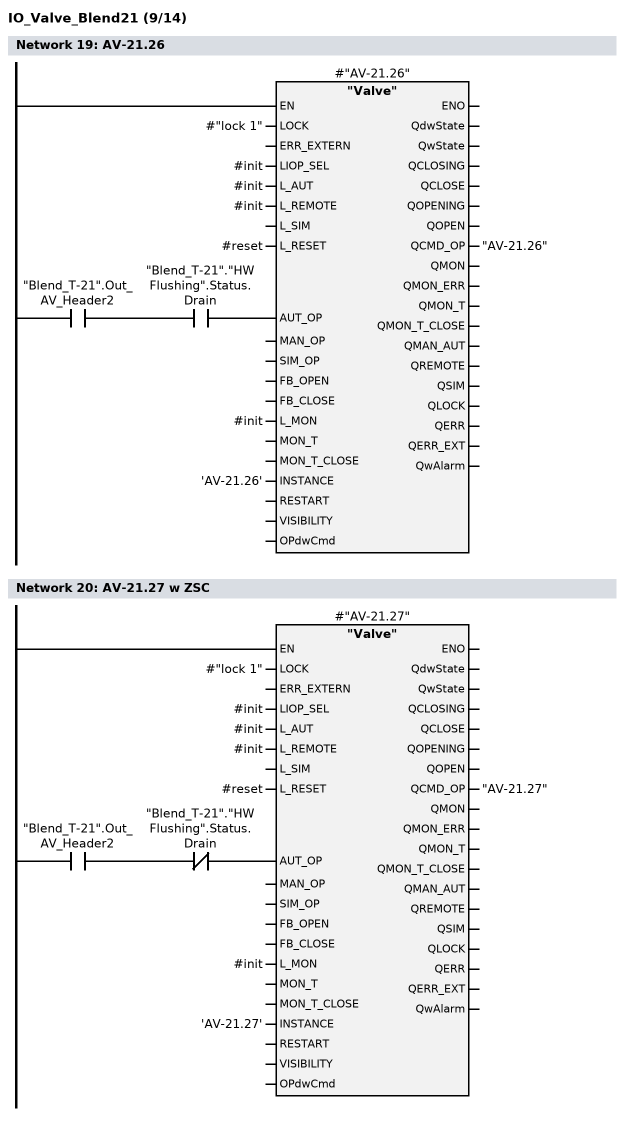
   RUNG wire#powerrail
      #"AV-21.26"(AUT_OP := wire#w1, LOCK := #"lock 1", ERR_EXTERN :=, LIOP_SEL := #init, L_AUT := #init, L_REMOTE := #init, L_SIM :=, L_RESET := #reset, MAN_OP :=, SIM_OP :=, FB_OPEN :=, FB_CLOSE :=, L_MON := #init, MON_T :=, MON_T_CLOSE :=, INSTANCE := 'AV-21.26', RESTART :=, VISIBILITY :=, OPdwCmd :=, QdwState =>, QwState =>, QCLOSING =>, QCLOSE =>, QOPENING =>, QOPEN =>, QCMD_OP => "AV-21.26", QMON =>, QMON_ERR =>, QMON_T =>, QMON_T_CLOSE =>, QMAN_AUT =>, QREMOTE =>, QSIM =>, QLOCK =>, QERR =>, QERR_EXT =>, QwAlarm =>)
   END_RUNG
   RUNG wire#powerrail
      Contact( "Blend_T-21".Out_AV_Header2 )
      Contact( "Blend_T-21"."HW Flushing".Status.Drain )
   END_RUNG wire#w1
   // the same network as SCL:
   #"AV-21.26"(LOCK := #"lock 1",   // "Valve"
               LIOP_SEL := #init,
               L_AUT := #init,
               L_REMOTE := #init,
               L_RESET := #reset,
               AUT_OP := "Blend_T-21".Out_AV_Header2 AND "Blend_T-21"."HW Flushing".Status.Drain,
               L_MON := #init,
               INSTANCE := 'AV-21.26',
               QCMD_OP => "AV-21.26");
END_REGION

REGION Network 20: AV-21.27 w ZSC
   RUNG wire#powerrail
      #"AV-21.27"(AUT_OP := wire#w1, LOCK := #"lock 1", ERR_EXTERN :=, LIOP_SEL := #init, L_AUT := #init, L_REMOTE := #init, L_SIM :=, L_RESET := #reset, MAN_OP :=, SIM_OP :=, FB_OPEN :=, FB_CLOSE :=, L_MON := #init, MON_T :=, MON_T_CLOSE :=, INSTANCE := 'AV-21.27', RESTART :=, VISIBILITY :=, OPdwCmd :=, QdwState =>, QwState =>, QCLOSING =>, QCLOSE =>, QOPENING =>, QOPEN =>, QCMD_OP => "AV-21.27", QMON =>, QMON_ERR =>, QMON_T =>, QMON_T_CLOSE =>, QMAN_AUT =>, QREMOTE =>, QSIM =>, QLOCK =>, QERR =>, QERR_EXT =>, QwAlarm =>)
   END_RUNG
   RUNG wire#powerrail
      Contact( "Blend_T-21".Out_AV_Header2 )
      I_Contact( "Blend_T-21"."HW Flushing".Status.Drain )
   END_RUNG wire#w1
   // the same network as SCL:
   #"AV-21.27"(LOCK := #"lock 1",   // "Valve"
               LIOP_SEL := #init,
               L_AUT := #init,
               L_REMOTE := #init,
               L_RESET := #reset,
               AUT_OP := "Blend_T-21".Out_AV_Header2 AND NOT "Blend_T-21"."HW Flushing".Status.Drain,
               L_MON := #init,
               INSTANCE := 'AV-21.27',
               QCMD_OP => "AV-21.27");
END_REGION

REGION Network 21: AV-21.28 w ZSC
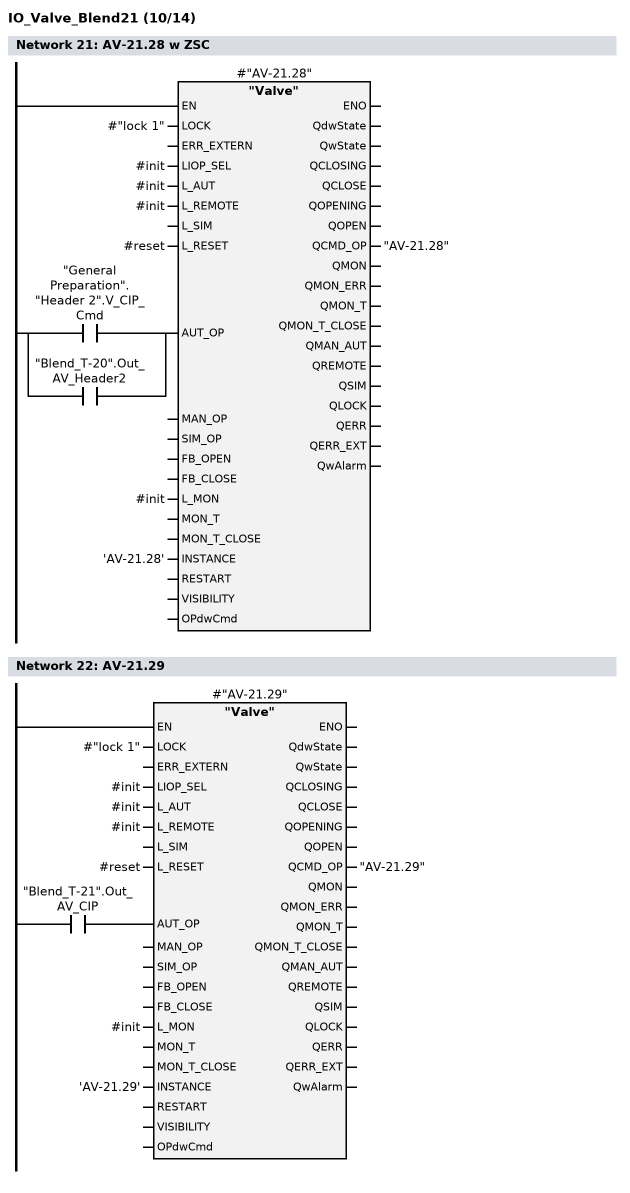
   RUNG wire#powerrail
      #"AV-21.28"(AUT_OP := wire#w1, LOCK := #"lock 1", ERR_EXTERN :=, LIOP_SEL := #init, L_AUT := #init, L_REMOTE := #init, L_SIM :=, L_RESET := #reset, MAN_OP :=, SIM_OP :=, FB_OPEN :=, FB_CLOSE :=, L_MON := #init, MON_T :=, MON_T_CLOSE :=, INSTANCE := 'AV-21.28', RESTART :=, VISIBILITY :=, OPdwCmd :=, QdwState =>, QwState =>, QCLOSING =>, QCLOSE =>, QOPENING =>, QOPEN =>, QCMD_OP => "AV-21.28", QMON =>, QMON_ERR =>, QMON_T =>, QMON_T_CLOSE =>, QMAN_AUT =>, QREMOTE =>, QSIM =>, QLOCK =>, QERR =>, QERR_EXT =>, QwAlarm =>)
   END_RUNG
   RUNG wire#powerrail
      Contact( "General Preparation"."Header 2".V_CIP_Cmd )
   END_RUNG wire#w1
   RUNG wire#powerrail
      Contact( "Blend_T-20".Out_AV_Header2 )
   END_RUNG wire#w1
   // the same network as SCL:
   #"AV-21.28"(LOCK := #"lock 1",   // "Valve"
               LIOP_SEL := #init,
               L_AUT := #init,
               L_REMOTE := #init,
               L_RESET := #reset,
               AUT_OP := "General Preparation"."Header 2".V_CIP_Cmd OR "Blend_T-20".Out_AV_Header2,
               L_MON := #init,
               INSTANCE := 'AV-21.28',
               QCMD_OP => "AV-21.28");
END_REGION

REGION Network 22: AV-21.29
   RUNG wire#powerrail
      #"AV-21.29"(AUT_OP := wire#w1, LOCK := #"lock 1", ERR_EXTERN :=, LIOP_SEL := #init, L_AUT := #init, L_REMOTE := #init, L_SIM :=, L_RESET := #reset, MAN_OP :=, SIM_OP :=, FB_OPEN :=, FB_CLOSE :=, L_MON := #init, MON_T :=, MON_T_CLOSE :=, INSTANCE := 'AV-21.29', RESTART :=, VISIBILITY :=, OPdwCmd :=, QdwState =>, QwState =>, QCLOSING =>, QCLOSE =>, QOPENING =>, QOPEN =>, QCMD_OP => "AV-21.29", QMON =>, QMON_ERR =>, QMON_T =>, QMON_T_CLOSE =>, QMAN_AUT =>, QREMOTE =>, QSIM =>, QLOCK =>, QERR =>, QERR_EXT =>, QwAlarm =>)
   END_RUNG
   RUNG wire#powerrail
      Contact( "Blend_T-21".Out_AV_CIP )
   END_RUNG wire#w1
   // the same network as SCL:
   #"AV-21.29"(LOCK := #"lock 1",   // "Valve"
               LIOP_SEL := #init,
               L_AUT := #init,
               L_REMOTE := #init,
               L_RESET := #reset,
               AUT_OP := "Blend_T-21".Out_AV_CIP,
               L_MON := #init,
               INSTANCE := 'AV-21.29',
               QCMD_OP => "AV-21.29");
END_REGION

REGION Network 23: AV-21.30
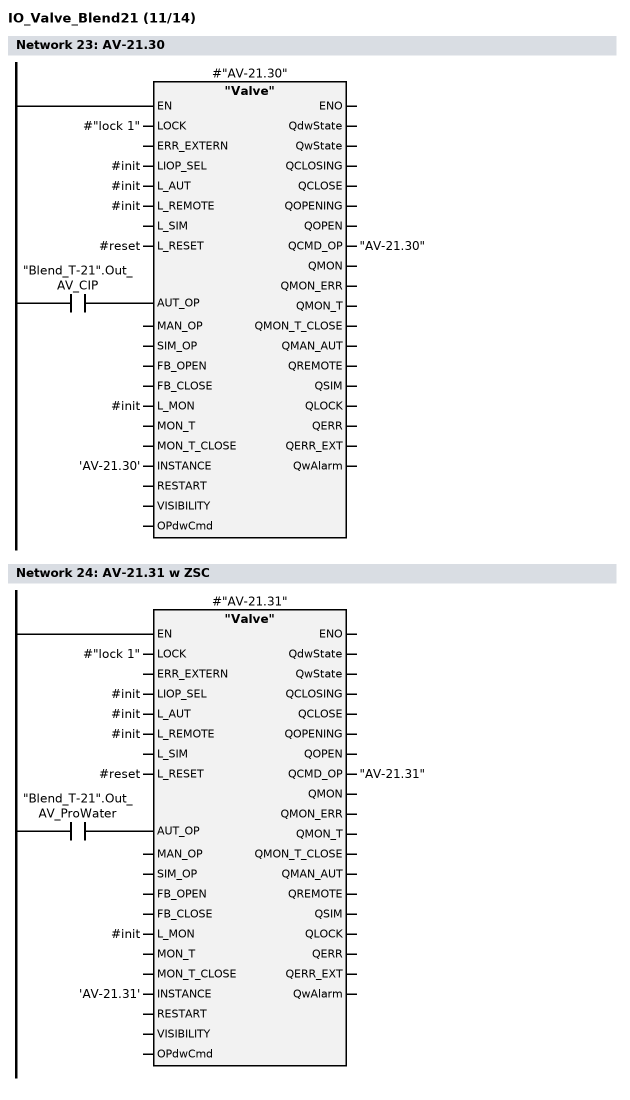
   RUNG wire#powerrail
      #"AV-21.30"(AUT_OP := wire#w1, LOCK := #"lock 1", ERR_EXTERN :=, LIOP_SEL := #init, L_AUT := #init, L_REMOTE := #init, L_SIM :=, L_RESET := #reset, MAN_OP :=, SIM_OP :=, FB_OPEN :=, FB_CLOSE :=, L_MON := #init, MON_T :=, MON_T_CLOSE :=, INSTANCE := 'AV-21.30', RESTART :=, VISIBILITY :=, OPdwCmd :=, QdwState =>, QwState =>, QCLOSING =>, QCLOSE =>, QOPENING =>, QOPEN =>, QCMD_OP => "AV-21.30", QMON =>, QMON_ERR =>, QMON_T =>, QMON_T_CLOSE =>, QMAN_AUT =>, QREMOTE =>, QSIM =>, QLOCK =>, QERR =>, QERR_EXT =>, QwAlarm =>)
   END_RUNG
   RUNG wire#powerrail
      Contact( "Blend_T-21".Out_AV_CIP )
   END_RUNG wire#w1
   // the same network as SCL:
   #"AV-21.30"(LOCK := #"lock 1",   // "Valve"
               LIOP_SEL := #init,
               L_AUT := #init,
               L_REMOTE := #init,
               L_RESET := #reset,
               AUT_OP := "Blend_T-21".Out_AV_CIP,
               L_MON := #init,
               INSTANCE := 'AV-21.30',
               QCMD_OP => "AV-21.30");
END_REGION

REGION Network 24: AV-21.31 w ZSC
   RUNG wire#powerrail
      #"AV-21.31"(AUT_OP := wire#w1, LOCK := #"lock 1", ERR_EXTERN :=, LIOP_SEL := #init, L_AUT := #init, L_REMOTE := #init, L_SIM :=, L_RESET := #reset, MAN_OP :=, SIM_OP :=, FB_OPEN :=, FB_CLOSE :=, L_MON := #init, MON_T :=, MON_T_CLOSE :=, INSTANCE := 'AV-21.31', RESTART :=, VISIBILITY :=, OPdwCmd :=, QdwState =>, QwState =>, QCLOSING =>, QCLOSE =>, QOPENING =>, QOPEN =>, QCMD_OP => "AV-21.31", QMON =>, QMON_ERR =>, QMON_T =>, QMON_T_CLOSE =>, QMAN_AUT =>, QREMOTE =>, QSIM =>, QLOCK =>, QERR =>, QERR_EXT =>, QwAlarm =>)
   END_RUNG
   RUNG wire#powerrail
      Contact( "Blend_T-21".Out_AV_ProWater )
   END_RUNG wire#w1
   // the same network as SCL:
   #"AV-21.31"(LOCK := #"lock 1",   // "Valve"
               LIOP_SEL := #init,
               L_AUT := #init,
               L_REMOTE := #init,
               L_RESET := #reset,
               AUT_OP := "Blend_T-21".Out_AV_ProWater,
               L_MON := #init,
               INSTANCE := 'AV-21.31',
               QCMD_OP => "AV-21.31");
END_REGION

REGION Network 25: AV-21.32 w ZSC
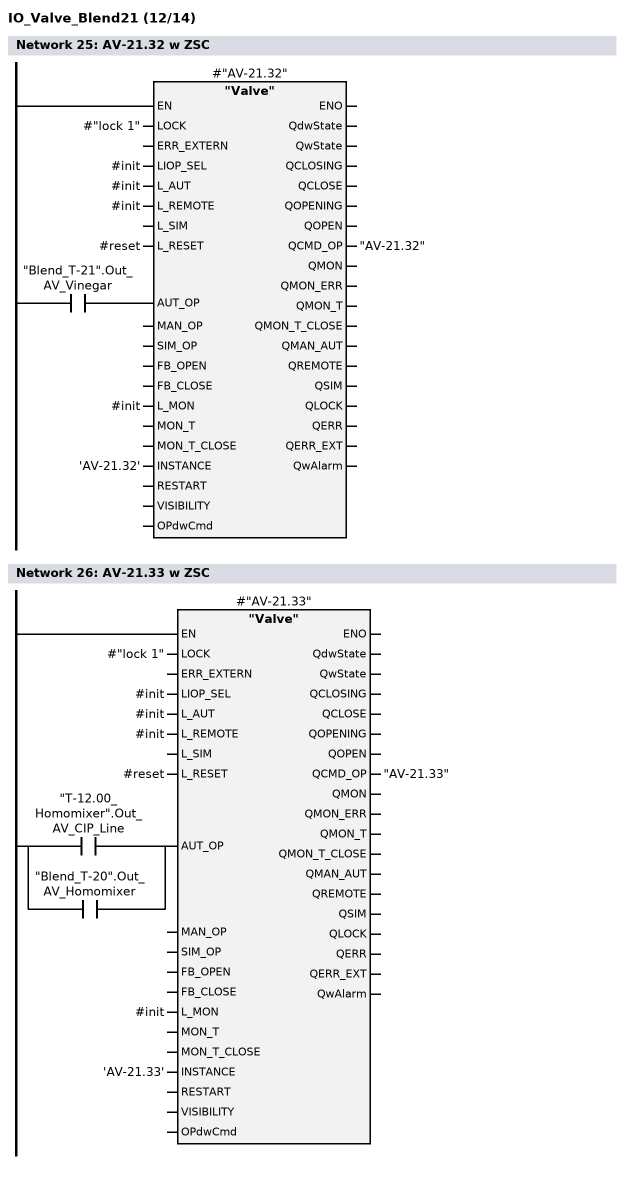
   RUNG wire#powerrail
      #"AV-21.32"(AUT_OP := wire#w1, LOCK := #"lock 1", ERR_EXTERN :=, LIOP_SEL := #init, L_AUT := #init, L_REMOTE := #init, L_SIM :=, L_RESET := #reset, MAN_OP :=, SIM_OP :=, FB_OPEN :=, FB_CLOSE :=, L_MON := #init, MON_T :=, MON_T_CLOSE :=, INSTANCE := 'AV-21.32', RESTART :=, VISIBILITY :=, OPdwCmd :=, QdwState =>, QwState =>, QCLOSING =>, QCLOSE =>, QOPENING =>, QOPEN =>, QCMD_OP => "AV-21.32", QMON =>, QMON_ERR =>, QMON_T =>, QMON_T_CLOSE =>, QMAN_AUT =>, QREMOTE =>, QSIM =>, QLOCK =>, QERR =>, QERR_EXT =>, QwAlarm =>)
   END_RUNG
   RUNG wire#powerrail
      Contact( "Blend_T-21".Out_AV_Vinegar )
   END_RUNG wire#w1
   // the same network as SCL:
   #"AV-21.32"(LOCK := #"lock 1",   // "Valve"
               LIOP_SEL := #init,
               L_AUT := #init,
               L_REMOTE := #init,
               L_RESET := #reset,
               AUT_OP := "Blend_T-21".Out_AV_Vinegar,
               L_MON := #init,
               INSTANCE := 'AV-21.32',
               QCMD_OP => "AV-21.32");
END_REGION

REGION Network 26: AV-21.33 w ZSC
   RUNG wire#powerrail
      #"AV-21.33"(AUT_OP := wire#w1, LOCK := #"lock 1", ERR_EXTERN :=, LIOP_SEL := #init, L_AUT := #init, L_REMOTE := #init, L_SIM :=, L_RESET := #reset, MAN_OP :=, SIM_OP :=, FB_OPEN :=, FB_CLOSE :=, L_MON := #init, MON_T :=, MON_T_CLOSE :=, INSTANCE := 'AV-21.33', RESTART :=, VISIBILITY :=, OPdwCmd :=, QdwState =>, QwState =>, QCLOSING =>, QCLOSE =>, QOPENING =>, QOPEN =>, QCMD_OP => "AV-21.33", QMON =>, QMON_ERR =>, QMON_T =>, QMON_T_CLOSE =>, QMAN_AUT =>, QREMOTE =>, QSIM =>, QLOCK =>, QERR =>, QERR_EXT =>, QwAlarm =>)
   END_RUNG
   RUNG wire#powerrail
      Contact( "T-12.00_Homomixer".Out_AV_CIP_Line )
   END_RUNG wire#w1
   RUNG wire#powerrail
      Contact( "Blend_T-20".Out_AV_Homomixer )
   END_RUNG wire#w1
   // the same network as SCL:
   #"AV-21.33"(LOCK := #"lock 1",   // "Valve"
               LIOP_SEL := #init,
               L_AUT := #init,
               L_REMOTE := #init,
               L_RESET := #reset,
               AUT_OP := "T-12.00_Homomixer".Out_AV_CIP_Line OR "Blend_T-20".Out_AV_Homomixer,
               L_MON := #init,
               INSTANCE := 'AV-21.33',
               QCMD_OP => "AV-21.33");
END_REGION

REGION Network 27: AV-21.34 w ZSC
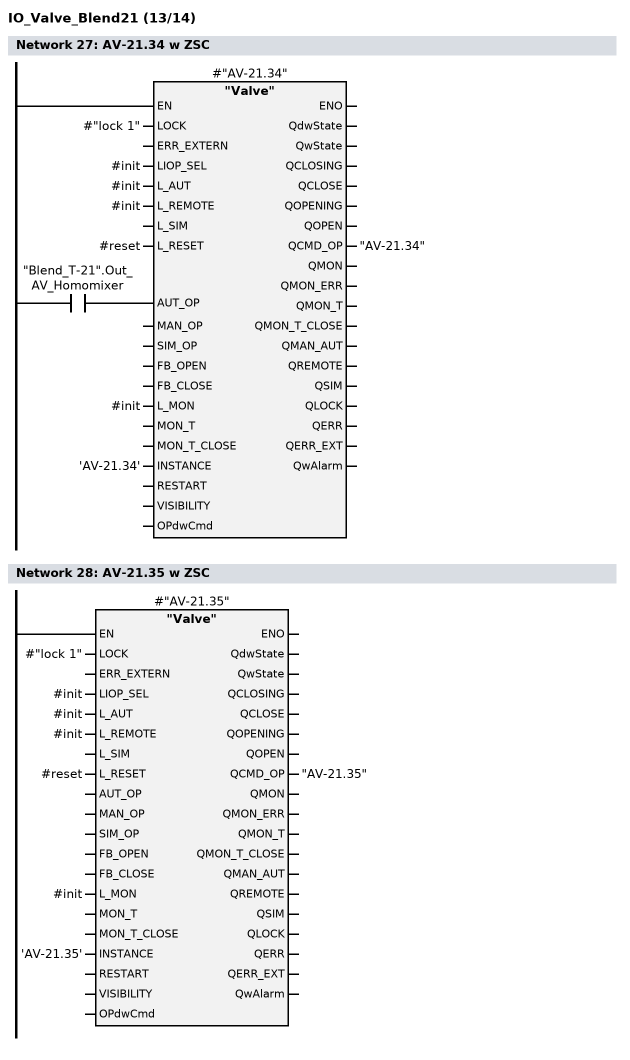
   RUNG wire#powerrail
      #"AV-21.34"(AUT_OP := wire#w1, LOCK := #"lock 1", ERR_EXTERN :=, LIOP_SEL := #init, L_AUT := #init, L_REMOTE := #init, L_SIM :=, L_RESET := #reset, MAN_OP :=, SIM_OP :=, FB_OPEN :=, FB_CLOSE :=, L_MON := #init, MON_T :=, MON_T_CLOSE :=, INSTANCE := 'AV-21.34', RESTART :=, VISIBILITY :=, OPdwCmd :=, QdwState =>, QwState =>, QCLOSING =>, QCLOSE =>, QOPENING =>, QOPEN =>, QCMD_OP => "AV-21.34", QMON =>, QMON_ERR =>, QMON_T =>, QMON_T_CLOSE =>, QMAN_AUT =>, QREMOTE =>, QSIM =>, QLOCK =>, QERR =>, QERR_EXT =>, QwAlarm =>)
   END_RUNG
   RUNG wire#powerrail
      Contact( "Blend_T-21".Out_AV_Homomixer )
   END_RUNG wire#w1
   // the same network as SCL:
   #"AV-21.34"(LOCK := #"lock 1",   // "Valve"
               LIOP_SEL := #init,
               L_AUT := #init,
               L_REMOTE := #init,
               L_RESET := #reset,
               AUT_OP := "Blend_T-21".Out_AV_Homomixer,
               L_MON := #init,
               INSTANCE := 'AV-21.34',
               QCMD_OP => "AV-21.34");
END_REGION

REGION Network 28: AV-21.35 w ZSC
   RUNG wire#powerrail
      #"AV-21.35"(LOCK := #"lock 1", ERR_EXTERN :=, LIOP_SEL := #init, L_AUT := #init, L_REMOTE := #init, L_SIM :=, L_RESET := #reset, AUT_OP :=, MAN_OP :=, SIM_OP :=, FB_OPEN :=, FB_CLOSE :=, L_MON := #init, MON_T :=, MON_T_CLOSE :=, INSTANCE := 'AV-21.35', RESTART :=, VISIBILITY :=, OPdwCmd :=, QdwState =>, QwState =>, QCLOSING =>, QCLOSE =>, QOPENING =>, QOPEN =>, QCMD_OP => "AV-21.35", QMON =>, QMON_ERR =>, QMON_T =>, QMON_T_CLOSE =>, QMAN_AUT =>, QREMOTE =>, QSIM =>, QLOCK =>, QERR =>, QERR_EXT =>, QwAlarm =>)
   END_RUNG
   // the same network as SCL:
   #"AV-21.35"(LOCK := #"lock 1",   // "Valve"
               LIOP_SEL := #init,
               L_AUT := #init,
               L_REMOTE := #init,
               L_RESET := #reset,
               L_MON := #init,
               INSTANCE := 'AV-21.35',
               QCMD_OP => "AV-21.35");
END_REGION

REGION Network 29: AV-21.41
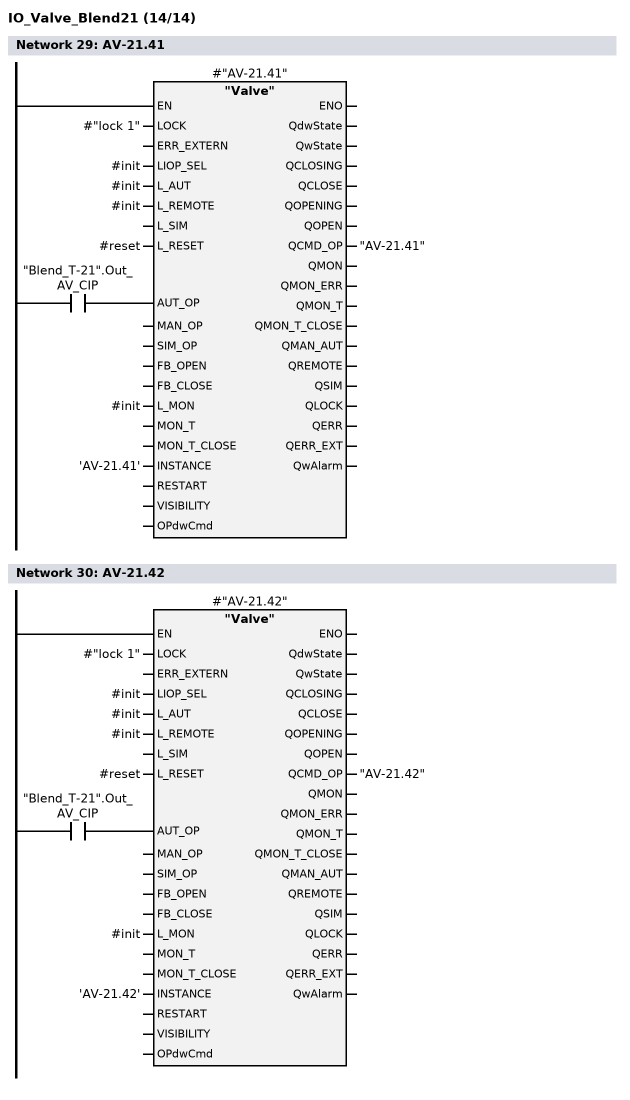
   RUNG wire#powerrail
      #"AV-21.41"(AUT_OP := wire#w1, LOCK := #"lock 1", ERR_EXTERN :=, LIOP_SEL := #init, L_AUT := #init, L_REMOTE := #init, L_SIM :=, L_RESET := #reset, MAN_OP :=, SIM_OP :=, FB_OPEN :=, FB_CLOSE :=, L_MON := #init, MON_T :=, MON_T_CLOSE :=, INSTANCE := 'AV-21.41', RESTART :=, VISIBILITY :=, OPdwCmd :=, QdwState =>, QwState =>, QCLOSING =>, QCLOSE =>, QOPENING =>, QOPEN =>, QCMD_OP => "AV-21.41", QMON =>, QMON_ERR =>, QMON_T =>, QMON_T_CLOSE =>, QMAN_AUT =>, QREMOTE =>, QSIM =>, QLOCK =>, QERR =>, QERR_EXT =>, QwAlarm =>)
   END_RUNG
   RUNG wire#powerrail
      Contact( "Blend_T-21".Out_AV_CIP )
   END_RUNG wire#w1
   // the same network as SCL:
   #"AV-21.41"(LOCK := #"lock 1",   // "Valve"
               LIOP_SEL := #init,
               L_AUT := #init,
               L_REMOTE := #init,
               L_RESET := #reset,
               AUT_OP := "Blend_T-21".Out_AV_CIP,
               L_MON := #init,
               INSTANCE := 'AV-21.41',
               QCMD_OP => "AV-21.41");
END_REGION

REGION Network 30: AV-21.42
   RUNG wire#powerrail
      #"AV-21.42"(AUT_OP := wire#w1, LOCK := #"lock 1", ERR_EXTERN :=, LIOP_SEL := #init, L_AUT := #init, L_REMOTE := #init, L_SIM :=, L_RESET := #reset, MAN_OP :=, SIM_OP :=, FB_OPEN :=, FB_CLOSE :=, L_MON := #init, MON_T :=, MON_T_CLOSE :=, INSTANCE := 'AV-21.42', RESTART :=, VISIBILITY :=, OPdwCmd :=, QdwState =>, QwState =>, QCLOSING =>, QCLOSE =>, QOPENING =>, QOPEN =>, QCMD_OP => "AV-21.42", QMON =>, QMON_ERR =>, QMON_T =>, QMON_T_CLOSE =>, QMAN_AUT =>, QREMOTE =>, QSIM =>, QLOCK =>, QERR =>, QERR_EXT =>, QwAlarm =>)
   END_RUNG
   RUNG wire#powerrail
      Contact( "Blend_T-21".Out_AV_CIP )
   END_RUNG wire#w1
   // the same network as SCL:
   #"AV-21.42"(LOCK := #"lock 1",   // "Valve"
               LIOP_SEL := #init,
               L_AUT := #init,
               L_REMOTE := #init,
               L_RESET := #reset,
               AUT_OP := "Blend_T-21".Out_AV_CIP,
               L_MON := #init,
               INSTANCE := 'AV-21.42',
               QCMD_OP => "AV-21.42");
END_REGION
END_FUNCTION_BLOCK
